(* PLC project Blank Project, Blank Blank 1.0 *)
(* stored: creationDateTime 2016-05-18T21:14:07, modificationDateTime 2017-02-16T14:47:06 *)

PROGRAM My_Program
  VAR
    transformer AT %QX0.0 : BOOL := 1;
    switch1 AT %QW0 : INT := 1;
    switch2 AT %QW1 : INT := 1;
    switch3 AT %QW2 : INT := 1;
    switch4 AT %QW3 : INT := 0;
    switch5 AT %QW4 : INT := 1;
    switch6 AT %QW5 : INT := 0;
  END_VAR

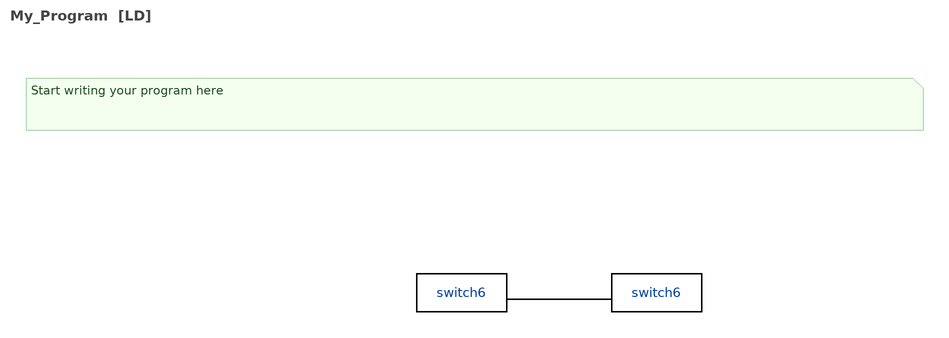
(* LD diagram, written out as Structured Text *)
(* Start writing your program here *)
switch6 := switch6;
END_PROGRAM

CONFIGURATION Config0
  RESOURCE Res0 ON PLC
    TASK TaskMain(INTERVAL := T#50ms, PRIORITY := 0);
    PROGRAM Inst0 WITH TaskMain : My_Program;
  END_RESOURCE
END_CONFIGURATION
